# EPICS IOC start-up script: test/startup/st.pneumatic-MCU031-CI0021330.iocsh
epicsEnvSet("MOTOR_PORT",      "$(SM_MOTOR_PORT=MCU1)")
#
epicsEnvSet("IPADDR",          "$(SM_IPADDR=CI0021330.esss.lu.se)")
epicsEnvSet("IPPORT",          "$(SM_IPPORT=48898)")
epicsEnvSet("ASYN_PORT",       "$(SM_ASYN_PORT=MC_CPU1)")
epicsEnvSet("AMSNETIDIOC",     "172.30.38.12.1.1")
epicsEnvSet("P",               "Labs-MCAG:MC-MCU-031:")
epicsEnvSet("R",               "")
epicsEnvSet("PREC",            "$(SM_PREC=3)")
epicsEnvSet("SM_NOAXES",       "3")
epicsEnvSet("ECM_OPTIONS",     "adsPort=852;amsNetIdRemote=10.0.7.5.1.1:852;amsNetIdLocal=$(AMSNETIDIOC)"

# No poller yet, see ethercatmcStartPoller at the end of the script
epicsEnvSet("ECM_MOVINGPOLLPERIOD", "0")
epicsEnvSet("ECM_IDLEPOLLPERIOD", "0")
< ethercatmcController.iocsh

#
# Axis 1, Shutter
#
epicsEnvSet("AXISCONFIG",      "")
epicsEnvSet("R",               "Shutter")
epicsEnvSet("AXIS_NO",         "1")
epicsEnvSet("DESC",            "$(SM_DESC=DESC)")
epicsEnvSet("EGU",             "$(SM_EGU=EGU)")
epicsEnvSet("R",               "Shutter-")
< ethercatmcShutter.iocsh

# Pressure
epicsEnvSet("P",               "$(P)Shutter-")
epicsEnvSet("R",               "Pressure")
epicsEnvSet("CHNO",            "1")
epicsEnvSet("ASYNPARAMNAME",   "Pressure")
epicsEnvSet("DESC",            "$(ASYNPARAMNAME)")
epicsEnvSet("PREC",            2)
epicsEnvSet("EGU",             "bar")
epicsEnvSet("SMOO",            0.5)
epicsEnvSet("ADEL",            0.05)
epicsEnvSet("MDEL",            0.05)
< ethercatmcAnalogInputSmooAdelMdel.iocsh
#< ethercatmcAnalogInput.iocsh

# Start polling, values are in millisconds
#
epicsEnvSet("MOVINGPOLLPERIOD", "200")
epicsEnvSet("IDLEPOLLPERIOD",  "500")
ethercatmcStartPoller("$(MOTOR_PORT)", "$(MOVINGPOLLPERIOD)", "$(IDLEPOLLPERIOD)")
